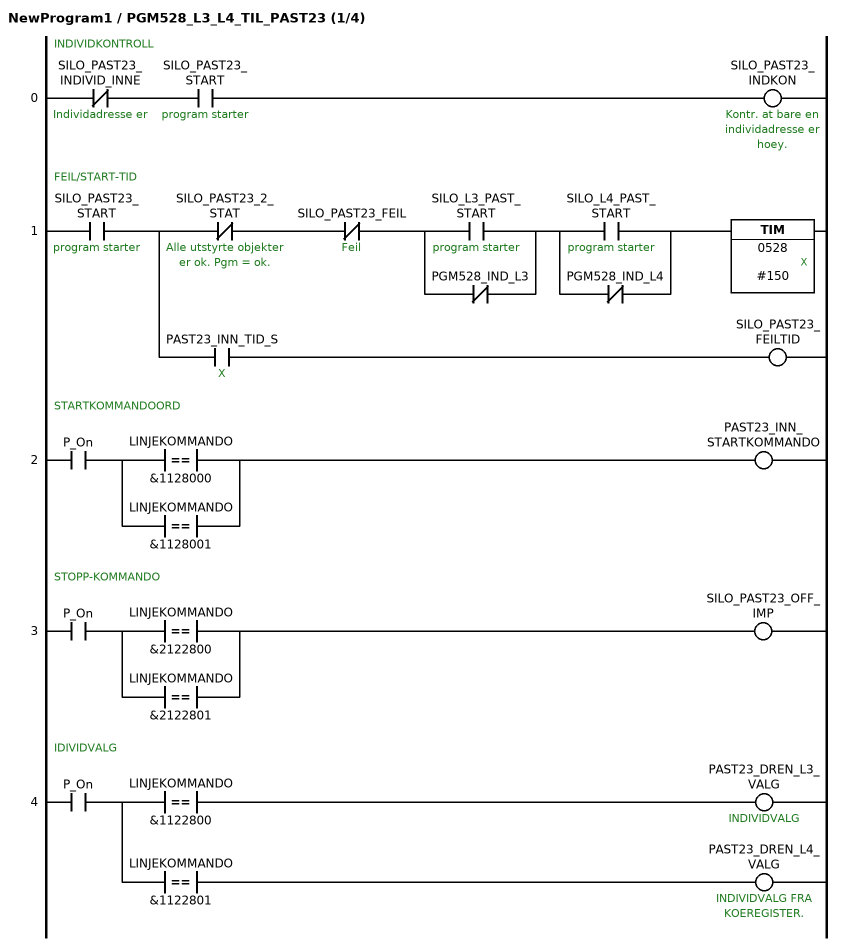
; [picture p696: NewProgram1 / PGM528_L3_L4_TIL_PAST23, rungs 0-4]
; rung 0: INDIVIDKONTROLL
LDNOT SILO_PAST23_INDIVID_INNE  ; Individadresse er
AND SILO_PAST23_START  ; program starter
OUT SILO_PAST23_INDKON  ; Kontr. at bare en individadresse er hoey.
; rung 1: FEIL/START-TID
LD SILO_PAST23_START  ; program starter
OUT TR0
ANDNOT SILO_PAST23_2_STAT  ; Alle utstyrte objekter er ok. Pgm = ok.
ANDNOT SILO_PAST23_FEIL  ; Feil
LD SILO_L3_PAST_START  ; program starter
ORNOT PGM528_IND_L3
ANDLD
LD SILO_L4_PAST_START  ; program starter
ORNOT PGM528_IND_L4
ANDLD
TIM 0528 #150  ; X
LD TR0
AND PAST23_INN_TID_S  ; X
OUT SILO_PAST23_FEILTID
; rung 2: STARTKOMMANDOORD
LD P_On
LD=L(301) LINJEKOMMANDO &1128000
OR=L(301) LINJEKOMMANDO &1128001
ANDLD
OUT PAST23_INN_STARTKOMMANDO
; rung 3: STOPP-KOMMANDO
LD P_On
LD=L(301) LINJEKOMMANDO &2122800
OR=L(301) LINJEKOMMANDO &2122801
ANDLD
OUT SILO_PAST23_OFF_IMP
; rung 4: IDIVIDVALG
LD P_On
OUT TR0
AND=L(301) LINJEKOMMANDO &1122800
OUT PAST23_DREN_L3_VALG  ; INDIVIDVALG
LD TR0
AND=L(301) LINJEKOMMANDO &1122801
OUT PAST23_DREN_L4_VALG  ; INDIVIDVALG FRA KOEREGISTER.

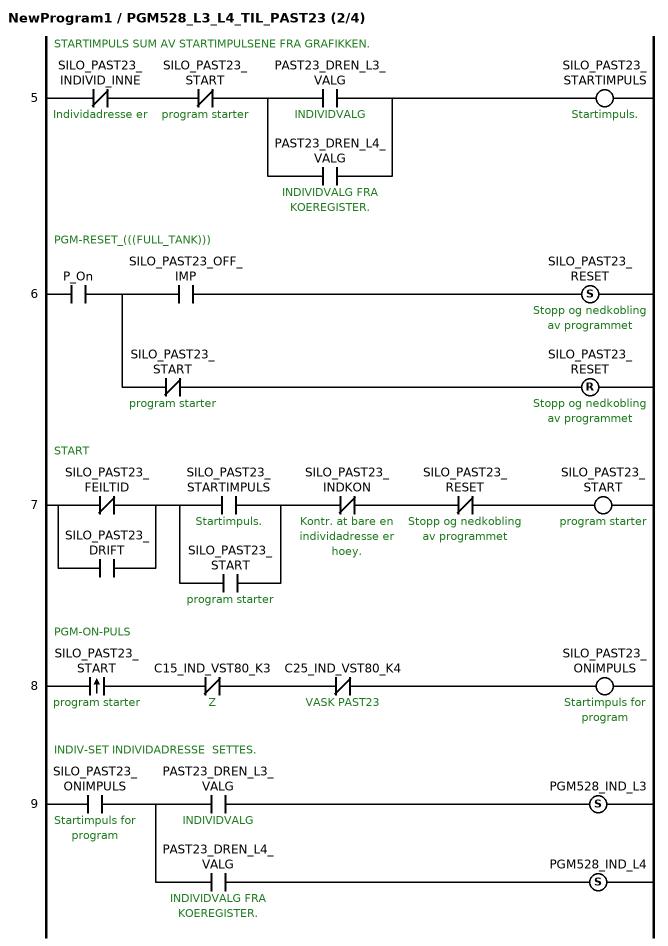
; rung 5: STARTIMPULS SUM AV STARTIMPULSENE FRA GRAFIKKEN.
LDNOT SILO_PAST23_INDIVID_INNE  ; Individadresse er
ANDNOT SILO_PAST23_START  ; program starter
LD PAST23_DREN_L3_VALG  ; INDIVIDVALG
OR PAST23_DREN_L4_VALG  ; INDIVIDVALG FRA KOEREGISTER.
ANDLD
OUT SILO_PAST23_STARTIMPULS  ; Startimpuls.
; rung 6: PGM-RESET_(((FULL_TANK)))
LD P_On
OUT TR0
AND SILO_PAST23_OFF_IMP
SET SILO_PAST23_RESET  ; Stopp og nedkobling av programmet
LD TR0
ANDNOT SILO_PAST23_START  ; program starter
RSET SILO_PAST23_RESET  ; Stopp og nedkobling av programmet
; rung 7: START
LDNOT SILO_PAST23_FEILTID
OR SILO_PAST23_DRIFT
LD SILO_PAST23_STARTIMPULS  ; Startimpuls.
OR SILO_PAST23_START  ; program starter
ANDLD
ANDNOT SILO_PAST23_INDKON  ; Kontr. at bare en individadresse er hoey.
ANDNOT SILO_PAST23_RESET  ; Stopp og nedkobling av programmet
OUT SILO_PAST23_START  ; program starter
; rung 8: PGM-ON-PULS
@LD SILO_PAST23_START  ; program starter
ANDNOT C15_IND_VST80_K3  ; Z
ANDNOT C25_IND_VST80_K4  ; VASK PAST23
OUT SILO_PAST23_ONIMPULS  ; Startimpuls for  program
; rung 9: INDIV-SET INDIVIDADRESSE  SETTES.
LD SILO_PAST23_ONIMPULS  ; Startimpuls for  program
OUT TR0
AND PAST23_DREN_L3_VALG  ; INDIVIDVALG
SET PGM528_IND_L3
LD TR0
AND PAST23_DREN_L4_VALG  ; INDIVIDVALG FRA KOEREGISTER.
SET PGM528_IND_L4

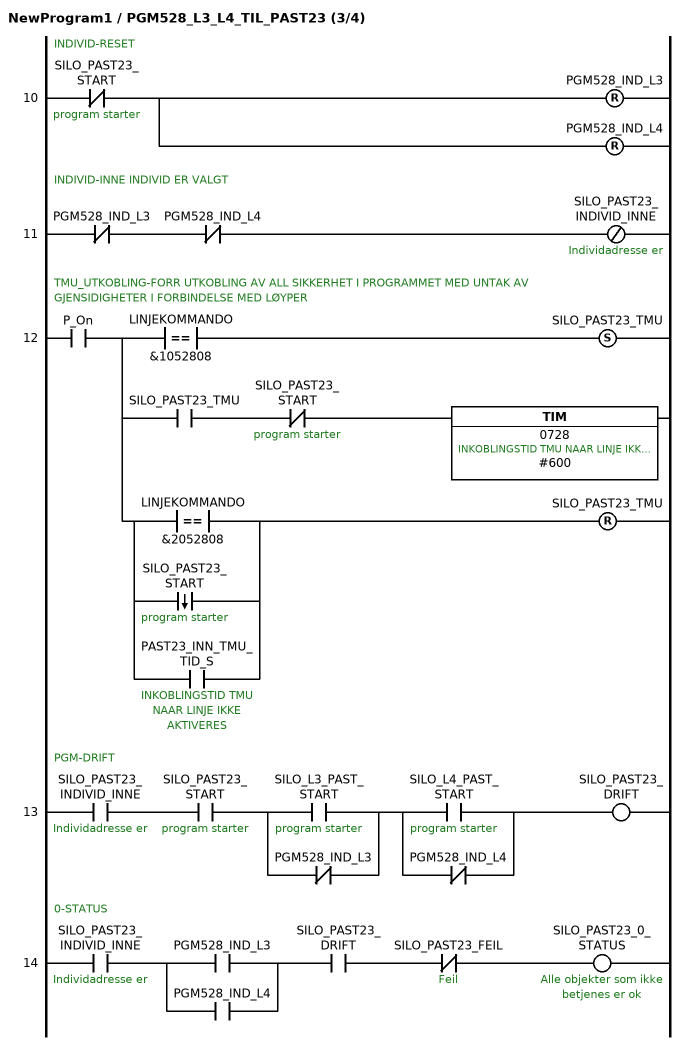
; rung 10: INDIVID-RESET
LDNOT SILO_PAST23_START  ; program starter
RSET PGM528_IND_L3
RSET PGM528_IND_L4
; rung 11: INDIVID-INNE INDIVID ER VALGT
LDNOT PGM528_IND_L3
ANDNOT PGM528_IND_L4
OUTNOT SILO_PAST23_INDIVID_INNE  ; Individadresse er
; rung 12: TMU_UTKOBLING-FORR UTKOBLING AV ALL SIKKERHET I PROGRAMMET MED UNTAK AV GJENSIDIGHETER I FORBINDELSE MED LØYPER
LD P_On
OUT TR0
AND=L(301) LINJEKOMMANDO &1052808
SET SILO_PAST23_TMU
LD TR0
AND SILO_PAST23_TMU
ANDNOT SILO_PAST23_START  ; program starter
TIM 0728 #600  ; INKOBLINGSTID TMU NAAR LINJE IKKE AKTIVERES
LD TR0
LD=L(301) LINJEKOMMANDO &2052808
%OR SILO_PAST23_START  ; program starter
OR PAST23_INN_TMU_TID_S  ; INKOBLINGSTID TMU NAAR LINJE IKKE AKTIVERES
ANDLD
RSET SILO_PAST23_TMU
; rung 13: PGM-DRIFT
LD SILO_PAST23_INDIVID_INNE  ; Individadresse er
AND SILO_PAST23_START  ; program starter
LD SILO_L3_PAST_START  ; program starter
ORNOT PGM528_IND_L3
ANDLD
LD SILO_L4_PAST_START  ; program starter
ORNOT PGM528_IND_L4
ANDLD
OUT SILO_PAST23_DRIFT
; rung 14: 0-STATUS
LD SILO_PAST23_INDIVID_INNE  ; Individadresse er
LD PGM528_IND_L3
OR PGM528_IND_L4
ANDLD
AND SILO_PAST23_DRIFT
ANDNOT SILO_PAST23_FEIL  ; Feil
OUT SILO_PAST23_0_STATUS  ; Alle objekter som ikke betjenes er ok

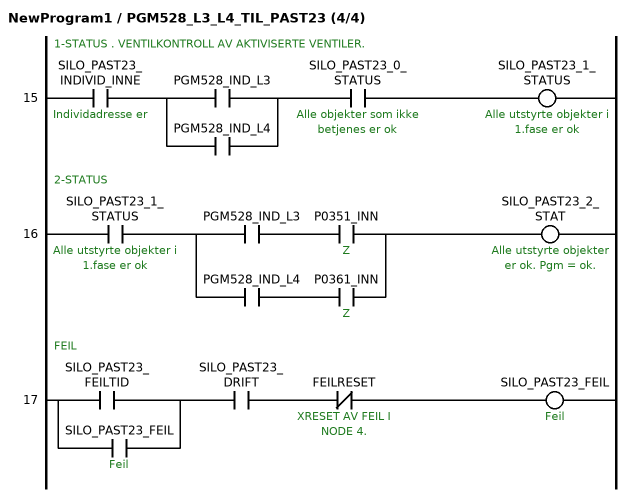
; rung 15: 1-STATUS . VENTILKONTROLL AV AKTIVISERTE VENTILER.
LD SILO_PAST23_INDIVID_INNE  ; Individadresse er
LD PGM528_IND_L3
OR PGM528_IND_L4
ANDLD
AND SILO_PAST23_0_STATUS  ; Alle objekter som ikke betjenes er ok
OUT SILO_PAST23_1_STATUS  ; Alle utstyrte objekter i 1.fase er ok
; rung 16: 2-STATUS
LD SILO_PAST23_1_STATUS  ; Alle utstyrte objekter i 1.fase er ok
LD PGM528_IND_L3
AND P0351_INN  ; Z
LD PGM528_IND_L4
AND P0361_INN  ; Z
ORLD
ANDLD
OUT SILO_PAST23_2_STAT  ; Alle utstyrte objekter er ok. Pgm = ok.
; rung 17: FEIL
LD SILO_PAST23_FEILTID
OR SILO_PAST23_FEIL  ; Feil
AND SILO_PAST23_DRIFT
ANDNOT FEILRESET  ; XRESET AV FEIL I NODE 4.
OUT SILO_PAST23_FEIL  ; Feil

### Section PGM529_T24_CONTAINER_TIL_PAST23

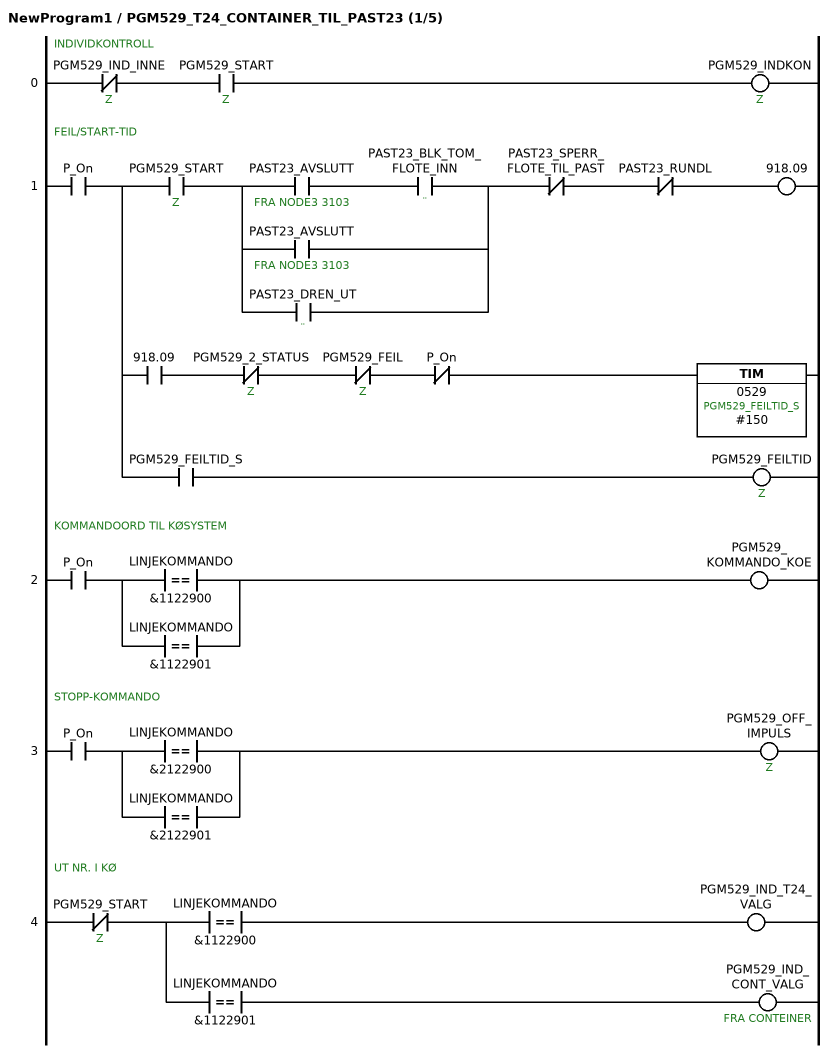
; rung 0: INDIVIDKONTROLL
LDNOT PGM529_IND_INNE  ; Z
AND PGM529_START  ; Z
OUT PGM529_INDKON  ; Z
; rung 1: FEIL/START-TID
LD P_On
OUT TR0
AND PGM529_START  ; Z
LD PAST23_AVSLUTT  ; FRA NODE3 3103
AND PAST23_BLK_TOM_FLOTE_INN  ; ¨
OR PAST23_AVSLUTT  ; FRA NODE3 3103
OR PAST23_DREN_UT  ; ¨
ANDLD
ANDNOT PAST23_SPERR_FLOTE_TIL_PAST
ANDNOT PAST23_RUNDL
OUT 918.09
LD TR0
AND 918.09
ANDNOT PGM529_2_STATUS  ; Z
ANDNOT PGM529_FEIL  ; Z
ANDNOT P_On
TIM 0529 #150  ; PGM529_FEILTID_S
LD TR0
AND PGM529_FEILTID_S
OUT PGM529_FEILTID  ; Z
; rung 2: KOMMANDOORD TIL KØSYSTEM
LD P_On
LD=L(301) LINJEKOMMANDO &1122900
OR=L(301) LINJEKOMMANDO &1122901
ANDLD
OUT PGM529_KOMMANDO_KOE
; rung 3: STOPP-KOMMANDO
LD P_On
LD=L(301) LINJEKOMMANDO &2122900
OR=L(301) LINJEKOMMANDO &2122901
ANDLD
OUT PGM529_OFF_IMPULS  ; Z
; rung 4: UT NR. I KØ
LDNOT PGM529_START  ; Z
OUT TR0
AND=L(301) LINJEKOMMANDO &1122900
OUT PGM529_IND_T24_VALG
LD TR0
AND=L(301) LINJEKOMMANDO &1122901
OUT PGM529_IND_CONT_VALG  ; FRA CONTEINER

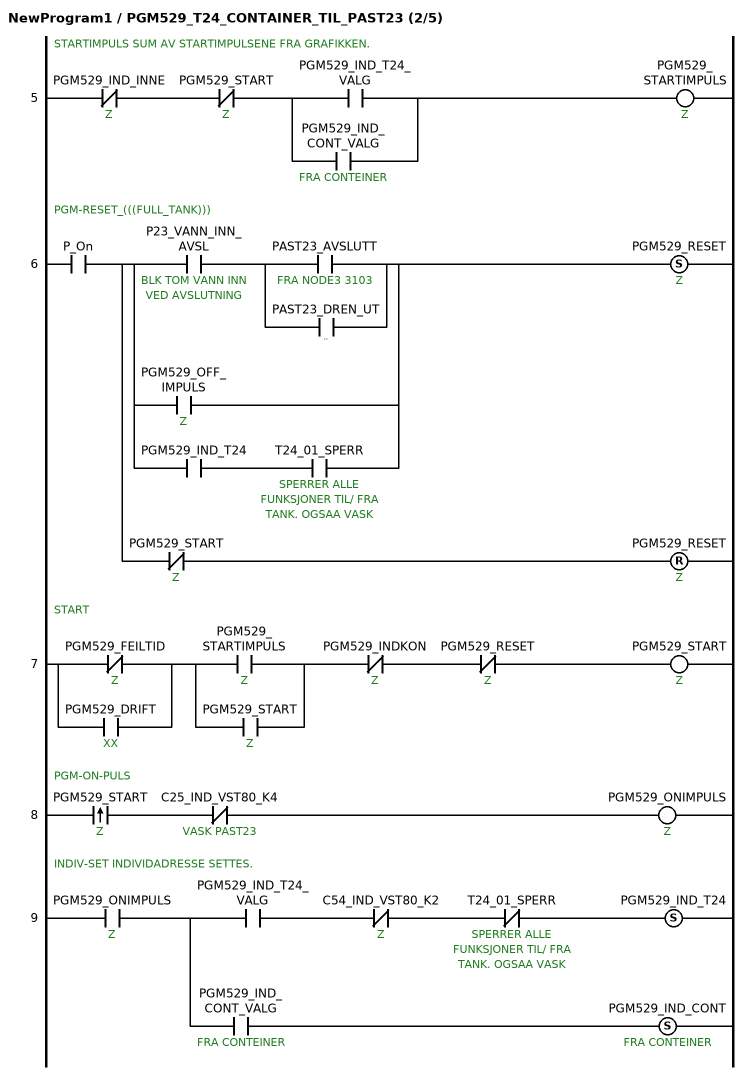
; rung 5: STARTIMPULS SUM AV STARTIMPULSENE FRA GRAFIKKEN.
LDNOT PGM529_IND_INNE  ; Z
ANDNOT PGM529_START  ; Z
LD PGM529_IND_T24_VALG
OR PGM529_IND_CONT_VALG  ; FRA CONTEINER
ANDLD
OUT PGM529_STARTIMPULS  ; Z
; rung 6: PGM-RESET_(((FULL_TANK)))
LD P_On
OUT TR0
LD P23_VANN_INN_AVSL  ; BLK TOM VANN INN VED AVSLUTNING
LD PAST23_AVSLUTT  ; FRA NODE3 3103
OR PAST23_DREN_UT  ; ¨
ANDLD
OR PGM529_OFF_IMPULS  ; Z
LD PGM529_IND_T24
AND T24_01_SPERR  ; SPERRER ALLE FUNKSJONER TIL/ FRA TANK. OGSAA VASK
ORLD
ANDLD
SET PGM529_RESET  ; Z
LD TR0
ANDNOT PGM529_START  ; Z
RSET PGM529_RESET  ; Z
; rung 7: START
LDNOT PGM529_FEILTID  ; Z
OR PGM529_DRIFT  ; XX
LD PGM529_STARTIMPULS  ; Z
OR PGM529_START  ; Z
ANDLD
ANDNOT PGM529_INDKON  ; Z
ANDNOT PGM529_RESET  ; Z
OUT PGM529_START  ; Z
; rung 8: PGM-ON-PULS
@LD PGM529_START  ; Z
ANDNOT C25_IND_VST80_K4  ; VASK PAST23
OUT PGM529_ONIMPULS  ; Z
; rung 9: INDIV-SET INDIVIDADRESSE SETTES.
LD PGM529_ONIMPULS  ; Z
OUT TR0
AND PGM529_IND_T24_VALG
ANDNOT C54_IND_VST80_K2  ; Z
ANDNOT T24_01_SPERR  ; SPERRER ALLE FUNKSJONER TIL/ FRA TANK. OGSAA VASK
SET PGM529_IND_T24
LD TR0
AND PGM529_IND_CONT_VALG  ; FRA CONTEINER
SET PGM529_IND_CONT  ; FRA CONTEINER

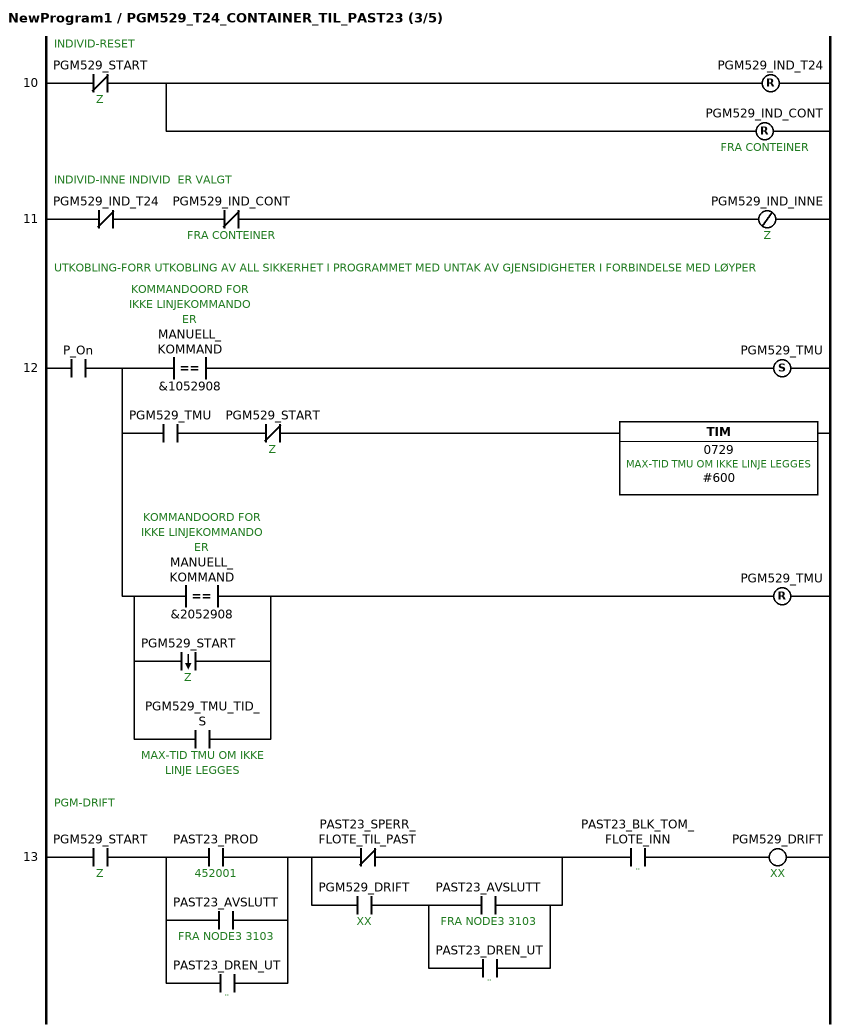
; rung 10: INDIVID-RESET
LDNOT PGM529_START  ; Z
RSET PGM529_IND_T24
RSET PGM529_IND_CONT  ; FRA CONTEINER
; rung 11: INDIVID-INNE INDIVID  ER VALGT
LDNOT PGM529_IND_T24
ANDNOT PGM529_IND_CONT  ; FRA CONTEINER
OUTNOT PGM529_IND_INNE  ; Z
; rung 12: UTKOBLING-FORR UTKOBLING AV ALL SIKKERHET I PROGRAMMET MED UNTAK AV GJENSIDIGHETER I FORBINDELSE MED LØYPER
LD P_On
OUT TR0
AND=L(301) MANUELL_KOMMAND &1052908  ; KOMMANDOORD FOR IKKE LINJEKOMMANDOER
SET PGM529_TMU
LD TR0
AND PGM529_TMU
ANDNOT PGM529_START  ; Z
TIM 0729 #600  ; MAX-TID TMU OM IKKE LINJE LEGGES
LD TR0
LD=L(301) MANUELL_KOMMAND &2052908  ; KOMMANDOORD FOR IKKE LINJEKOMMANDOER
%OR PGM529_START  ; Z
OR PGM529_TMU_TID_S  ; MAX-TID TMU OM IKKE LINJE LEGGES
ANDLD
RSET PGM529_TMU
; rung 13: PGM-DRIFT
LD PGM529_START  ; Z
LD PAST23_PROD  ; 452001
OR PAST23_AVSLUTT  ; FRA NODE3 3103
OR PAST23_DREN_UT  ; ¨
ANDLD
LDNOT PAST23_SPERR_FLOTE_TIL_PAST
LD PGM529_DRIFT  ; XX
LD PAST23_AVSLUTT  ; FRA NODE3 3103
OR PAST23_DREN_UT  ; ¨
ANDLD
ORLD
ANDLD
AND PAST23_BLK_TOM_FLOTE_INN  ; ¨
OUT PGM529_DRIFT  ; XX

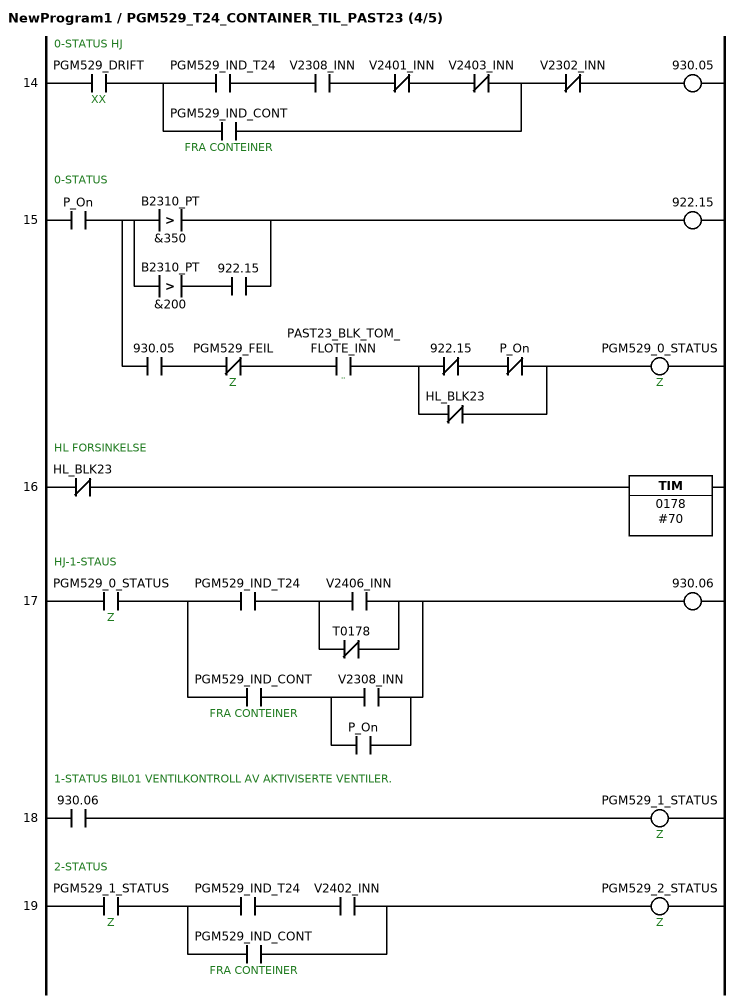
; rung 14: 0-STATUS HJ
LD PGM529_DRIFT  ; XX
LD PGM529_IND_T24
AND V2308_INN
ANDNOT V2401_INN
ANDNOT V2403_INN
OR PGM529_IND_CONT  ; FRA CONTEINER
ANDLD
ANDNOT V2302_INN
OUT 930.05
; rung 15: 0-STATUS
LD P_On
OUT TR0
LD>(320) B2310_PT &350
LD>(320) B2310_PT &200
AND 922.15
ORLD
ANDLD
OUT 922.15
LD TR0
AND 930.05
ANDNOT PGM529_FEIL  ; Z
AND PAST23_BLK_TOM_FLOTE_INN  ; ¨
LDNOT 922.15
ANDNOT P_On
ORNOT HL_BLK23
ANDLD
OUT PGM529_0_STATUS  ; Z
; rung 16: HL FORSINKELSE
LDNOT HL_BLK23
TIM 0178 #70
; rung 17: HJ-1-STAUS
LD PGM529_0_STATUS  ; Z
LD PGM529_IND_T24
LD V2406_INN
ORNOT T0178
ANDLD
LD PGM529_IND_CONT  ; FRA CONTEINER
LD V2308_INN
OR P_On
ANDLD
ORLD
ANDLD
OUT 930.06
; rung 18: 1-STATUS BIL01 VENTILKONTROLL AV AKTIVISERTE VENTILER.
LD 930.06
OUT PGM529_1_STATUS  ; Z
; rung 19: 2-STATUS
LD PGM529_1_STATUS  ; Z
LD PGM529_IND_T24
AND V2402_INN
OR PGM529_IND_CONT  ; FRA CONTEINER
ANDLD
OUT PGM529_2_STATUS  ; Z

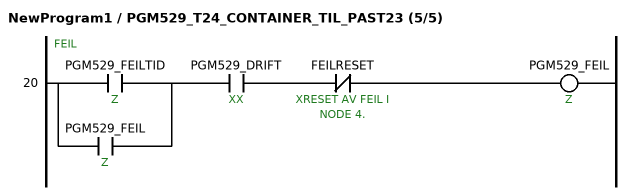
; rung 20: FEIL
LD PGM529_FEILTID  ; Z
OR PGM529_FEIL  ; Z
AND PGM529_DRIFT  ; XX
ANDNOT FEILRESET  ; XRESET AV FEIL I NODE 4.
OUT PGM529_FEIL  ; Z

### Section PGM584_TIL_T2740_2741

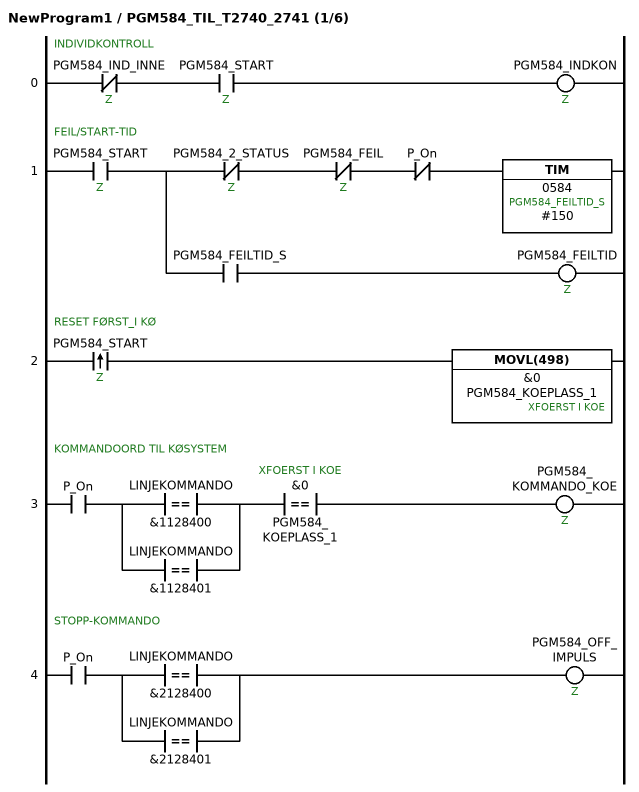
; rung 0: INDIVIDKONTROLL
LDNOT PGM584_IND_INNE  ; Z
AND PGM584_START  ; Z
OUT PGM584_INDKON  ; Z
; rung 1: FEIL/START-TID
LD PGM584_START  ; Z
OUT TR0
ANDNOT PGM584_2_STATUS  ; Z
ANDNOT PGM584_FEIL  ; Z
ANDNOT P_On
TIM 0584 #150  ; PGM584_FEILTID_S
LD TR0
AND PGM584_FEILTID_S
OUT PGM584_FEILTID  ; Z
; rung 2: RESET FØRST_I KØ
@LD PGM584_START  ; Z
MOVL(498) &0 PGM584_KOEPLASS_1  ; XFOERST I KOE
; rung 3: KOMMANDOORD TIL KØSYSTEM
LD P_On
LD=L(301) LINJEKOMMANDO &1128400
OR=L(301) LINJEKOMMANDO &1128401
ANDLD
AND=L(301) &0 PGM584_KOEPLASS_1  ; XFOERST I KOE
OUT PGM584_KOMMANDO_KOE  ; Z
; rung 4: STOPP-KOMMANDO
LD P_On
LD=L(301) LINJEKOMMANDO &2128400
OR=L(301) LINJEKOMMANDO &2128401
ANDLD
OUT PGM584_OFF_IMPULS  ; Z

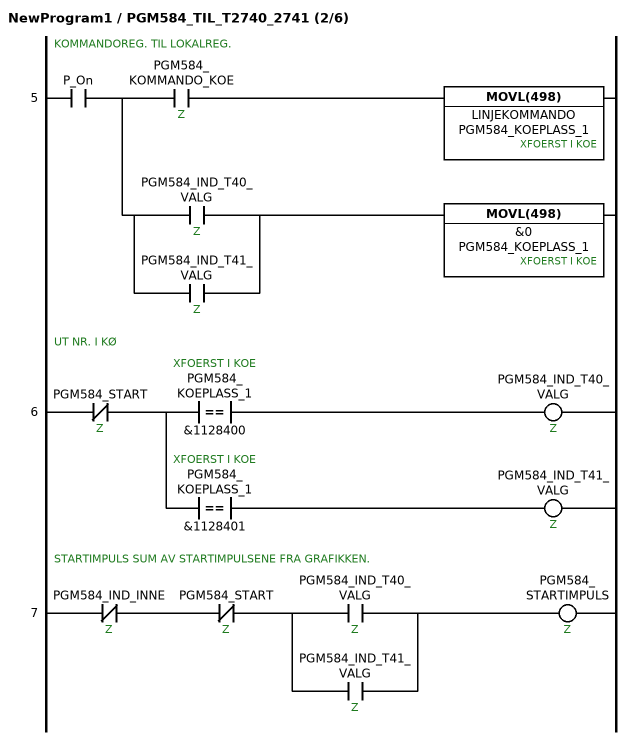
; rung 5: KOMMANDOREG. TIL LOKALREG.
LD P_On
OUT TR0
AND PGM584_KOMMANDO_KOE  ; Z
MOVL(498) LINJEKOMMANDO PGM584_KOEPLASS_1  ; XFOERST I KOE
LD TR0
LD PGM584_IND_T40_VALG  ; Z
OR PGM584_IND_T41_VALG  ; Z
ANDLD
MOVL(498) &0 PGM584_KOEPLASS_1  ; XFOERST I KOE
; rung 6: UT NR. I KØ
LDNOT PGM584_START  ; Z
OUT TR0
AND=L(301) PGM584_KOEPLASS_1 &1128400  ; XFOERST I KOE
OUT PGM584_IND_T40_VALG  ; Z
LD TR0
AND=L(301) PGM584_KOEPLASS_1 &1128401  ; XFOERST I KOE
OUT PGM584_IND_T41_VALG  ; Z
; rung 7: STARTIMPULS SUM AV STARTIMPULSENE FRA GRAFIKKEN.
LDNOT PGM584_IND_INNE  ; Z
ANDNOT PGM584_START  ; Z
LD PGM584_IND_T40_VALG  ; Z
OR PGM584_IND_T41_VALG  ; Z
ANDLD
OUT PGM584_STARTIMPULS  ; Z

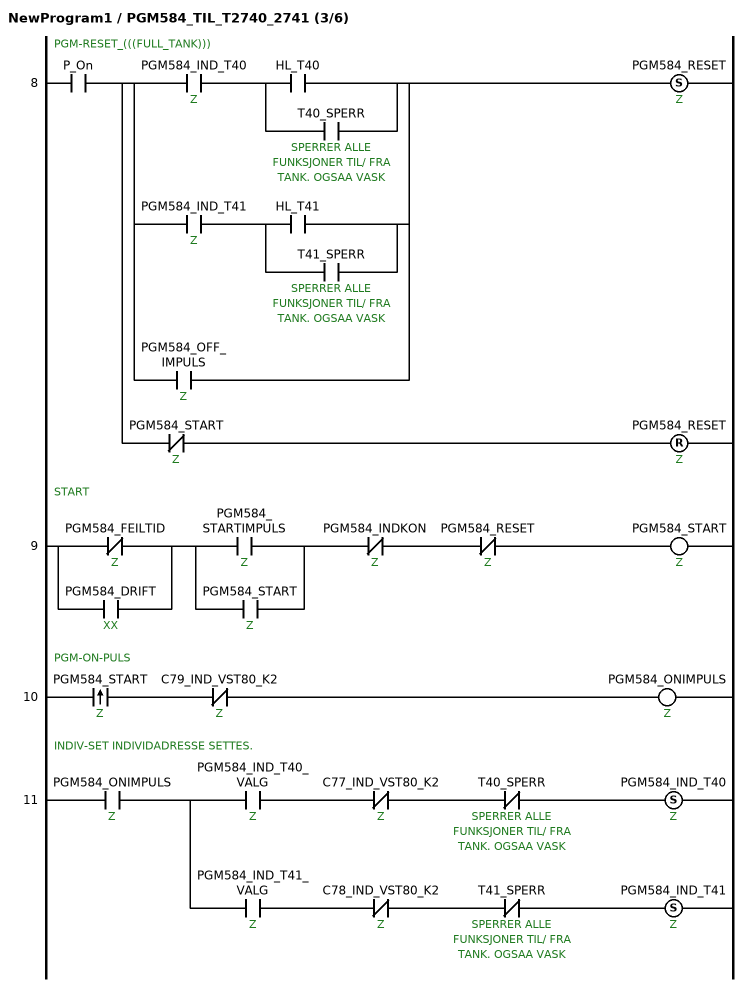
; rung 8: PGM-RESET_(((FULL_TANK)))
LD P_On
OUT TR0
LD PGM584_IND_T40  ; Z
LD HL_T40
OR T40_SPERR  ; SPERRER ALLE FUNKSJONER TIL/ FRA TANK. OGSAA VASK
ANDLD
LD PGM584_IND_T41  ; Z
LD HL_T41
OR T41_SPERR  ; SPERRER ALLE FUNKSJONER TIL/ FRA TANK. OGSAA VASK
ANDLD
ORLD
OR PGM584_OFF_IMPULS  ; Z
ANDLD
SET PGM584_RESET  ; Z
LD TR0
ANDNOT PGM584_START  ; Z
RSET PGM584_RESET  ; Z
; rung 9: START
LDNOT PGM584_FEILTID  ; Z
OR PGM584_DRIFT  ; XX
LD PGM584_STARTIMPULS  ; Z
OR PGM584_START  ; Z
ANDLD
ANDNOT PGM584_INDKON  ; Z
ANDNOT PGM584_RESET  ; Z
OUT PGM584_START  ; Z
; rung 10: PGM-ON-PULS
@LD PGM584_START  ; Z
ANDNOT C79_IND_VST80_K2  ; Z
OUT PGM584_ONIMPULS  ; Z
; rung 11: INDIV-SET INDIVIDADRESSE SETTES.
LD PGM584_ONIMPULS  ; Z
OUT TR0
AND PGM584_IND_T40_VALG  ; Z
ANDNOT C77_IND_VST80_K2  ; Z
ANDNOT T40_SPERR  ; SPERRER ALLE FUNKSJONER TIL/ FRA TANK. OGSAA VASK
SET PGM584_IND_T40  ; Z
LD TR0
AND PGM584_IND_T41_VALG  ; Z
ANDNOT C78_IND_VST80_K2  ; Z
ANDNOT T41_SPERR  ; SPERRER ALLE FUNKSJONER TIL/ FRA TANK. OGSAA VASK
SET PGM584_IND_T41  ; Z

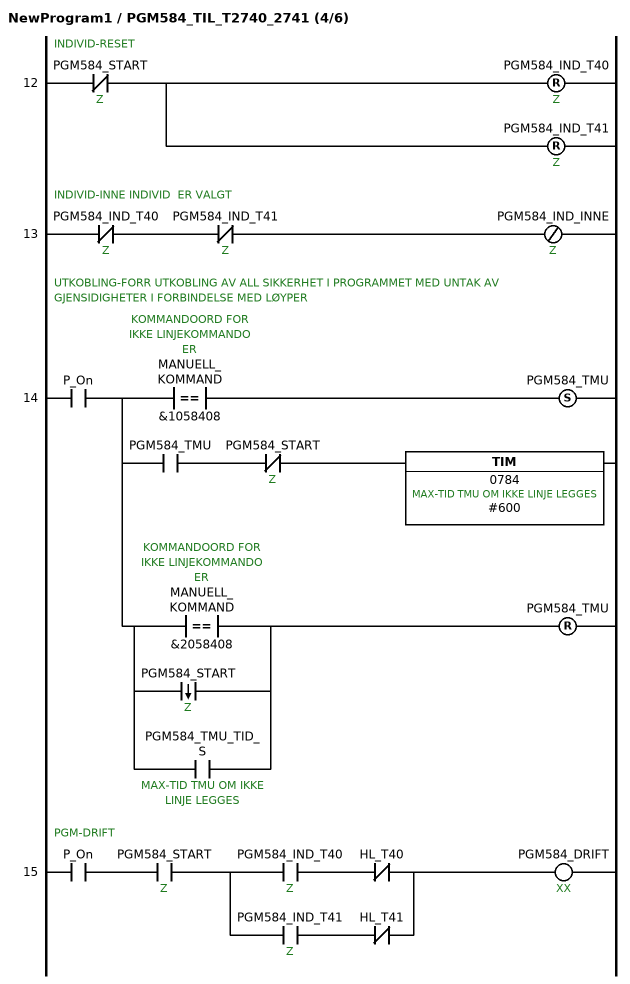
; rung 12: INDIVID-RESET
LDNOT PGM584_START  ; Z
RSET PGM584_IND_T40  ; Z
RSET PGM584_IND_T41  ; Z
; rung 13: INDIVID-INNE INDIVID  ER VALGT
LDNOT PGM584_IND_T40  ; Z
ANDNOT PGM584_IND_T41  ; Z
OUTNOT PGM584_IND_INNE  ; Z
; rung 14: UTKOBLING-FORR UTKOBLING AV ALL SIKKERHET I PROGRAMMET MED UNTAK AV GJENSIDIGHETER I FORBINDELSE MED LØYPER
LD P_On
OUT TR0
AND=L(301) MANUELL_KOMMAND &1058408  ; KOMMANDOORD FOR IKKE LINJEKOMMANDOER
SET PGM584_TMU
LD TR0
AND PGM584_TMU
ANDNOT PGM584_START  ; Z
TIM 0784 #600  ; MAX-TID TMU OM IKKE LINJE LEGGES
LD TR0
LD=L(301) MANUELL_KOMMAND &2058408  ; KOMMANDOORD FOR IKKE LINJEKOMMANDOER
%OR PGM584_START  ; Z
OR PGM584_TMU_TID_S  ; MAX-TID TMU OM IKKE LINJE LEGGES
ANDLD
RSET PGM584_TMU
; rung 15: PGM-DRIFT
LD P_On
AND PGM584_START  ; Z
LD PGM584_IND_T40  ; Z
ANDNOT HL_T40
LD PGM584_IND_T41  ; Z
ANDNOT HL_T41
ORLD
ANDLD
OUT PGM584_DRIFT  ; XX

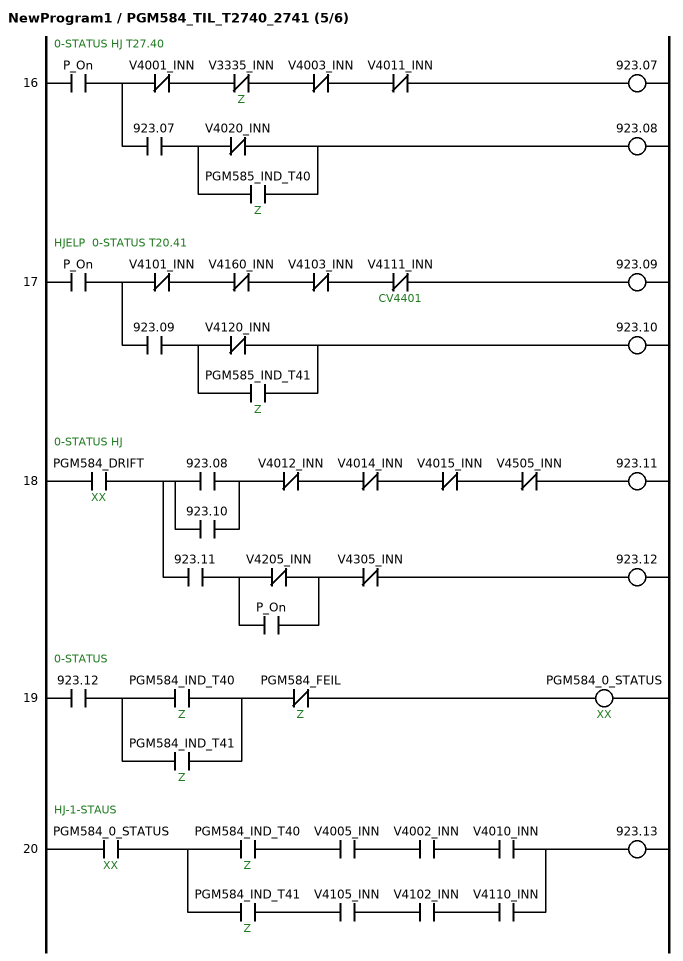
; rung 16: 0-STATUS HJ T27.40
LD P_On
OUT TR0
ANDNOT V4001_INN
ANDNOT V3335_INN  ; Z
ANDNOT V4003_INN
ANDNOT V4011_INN
OUT 923.07
LD TR0
AND 923.07
LDNOT V4020_INN
OR PGM585_IND_T40  ; Z
ANDLD
OUT 923.08
; rung 17: HJELP  0-STATUS T20.41
LD P_On
OUT TR0
ANDNOT V4101_INN
ANDNOT V4160_INN
ANDNOT V4103_INN
ANDNOT V4111_INN  ; CV4401
OUT 923.09
LD TR0
AND 923.09
LDNOT V4120_INN
OR PGM585_IND_T41  ; Z
ANDLD
OUT 923.10
; rung 18: 0-STATUS HJ
LD PGM584_DRIFT  ; XX
OUT TR0
LD 923.08
OR 923.10
ANDLD
ANDNOT V4012_INN
ANDNOT V4014_INN
ANDNOT V4015_INN
ANDNOT V4505_INN
OUT 923.11
LD TR0
AND 923.11
LDNOT V4205_INN
OR P_On
ANDLD
ANDNOT V4305_INN
OUT 923.12
; rung 19: 0-STATUS
LD 923.12
LD PGM584_IND_T40  ; Z
OR PGM584_IND_T41  ; Z
ANDLD
ANDNOT PGM584_FEIL  ; Z
OUT PGM584_0_STATUS  ; XX
; rung 20: HJ-1-STAUS
LD PGM584_0_STATUS  ; XX
LD PGM584_IND_T40  ; Z
AND V4005_INN
AND V4002_INN
AND V4010_INN
LD PGM584_IND_T41  ; Z
AND V4105_INN
AND V4102_INN
AND V4110_INN
ORLD
ANDLD
OUT 923.13

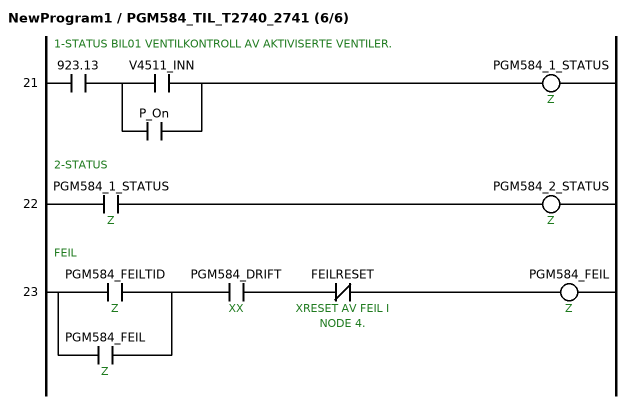
; rung 21: 1-STATUS BIL01 VENTILKONTROLL AV AKTIVISERTE VENTILER.
LD 923.13
LD V4511_INN
OR P_On
ANDLD
OUT PGM584_1_STATUS  ; Z
; rung 22: 2-STATUS
LD PGM584_1_STATUS  ; Z
OUT PGM584_2_STATUS  ; Z
; rung 23: FEIL
LD PGM584_FEILTID  ; Z
OR PGM584_FEIL  ; Z
AND PGM584_DRIFT  ; XX
ANDNOT FEILRESET  ; XRESET AV FEIL I NODE 4.
OUT PGM584_FEIL  ; Z

### Section PGM585_FRA_T2740_2741

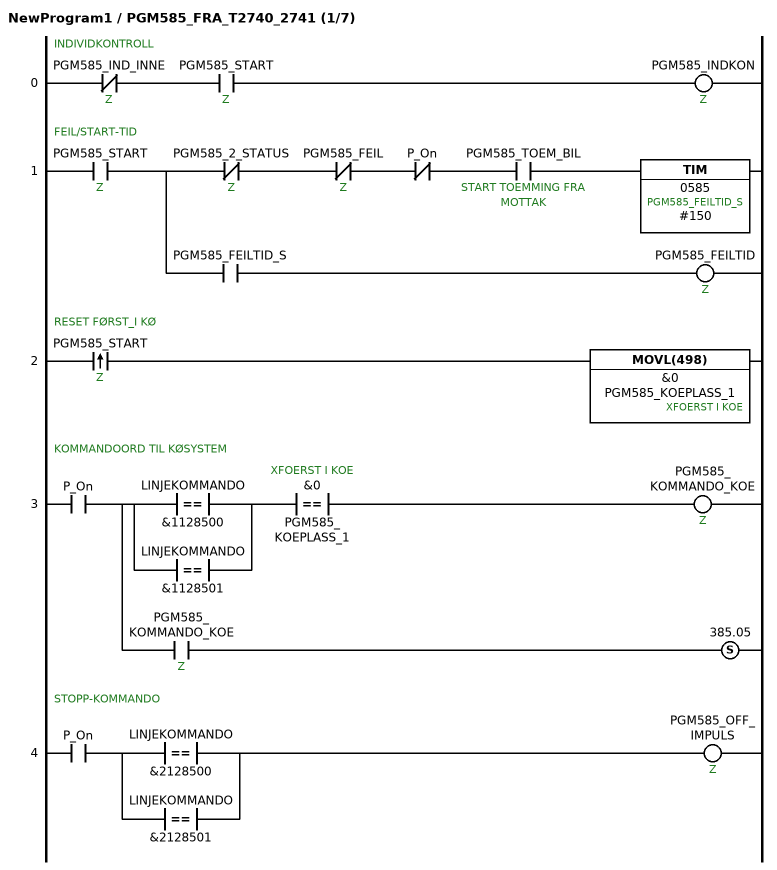
; rung 0: INDIVIDKONTROLL
LDNOT PGM585_IND_INNE  ; Z
AND PGM585_START  ; Z
OUT PGM585_INDKON  ; Z
; rung 1: FEIL/START-TID
LD PGM585_START  ; Z
OUT TR0
ANDNOT PGM585_2_STATUS  ; Z
ANDNOT PGM585_FEIL  ; Z
ANDNOT P_On
AND PGM585_TOEM_BIL  ; START TOEMMING FRA MOTTAK
TIM 0585 #150  ; PGM585_FEILTID_S
LD TR0
AND PGM585_FEILTID_S
OUT PGM585_FEILTID  ; Z
; rung 2: RESET FØRST_I KØ
@LD PGM585_START  ; Z
MOVL(498) &0 PGM585_KOEPLASS_1  ; XFOERST I KOE
; rung 3: KOMMANDOORD TIL KØSYSTEM
LD P_On
OUT TR0
LD=L(301) LINJEKOMMANDO &1128500
OR=L(301) LINJEKOMMANDO &1128501
ANDLD
AND=L(301) &0 PGM585_KOEPLASS_1  ; XFOERST I KOE
OUT PGM585_KOMMANDO_KOE  ; Z
LD TR0
AND PGM585_KOMMANDO_KOE  ; Z
SET 385.05
; rung 4: STOPP-KOMMANDO
LD P_On
LD=L(301) LINJEKOMMANDO &2128500
OR=L(301) LINJEKOMMANDO &2128501
ANDLD
OUT PGM585_OFF_IMPULS  ; Z

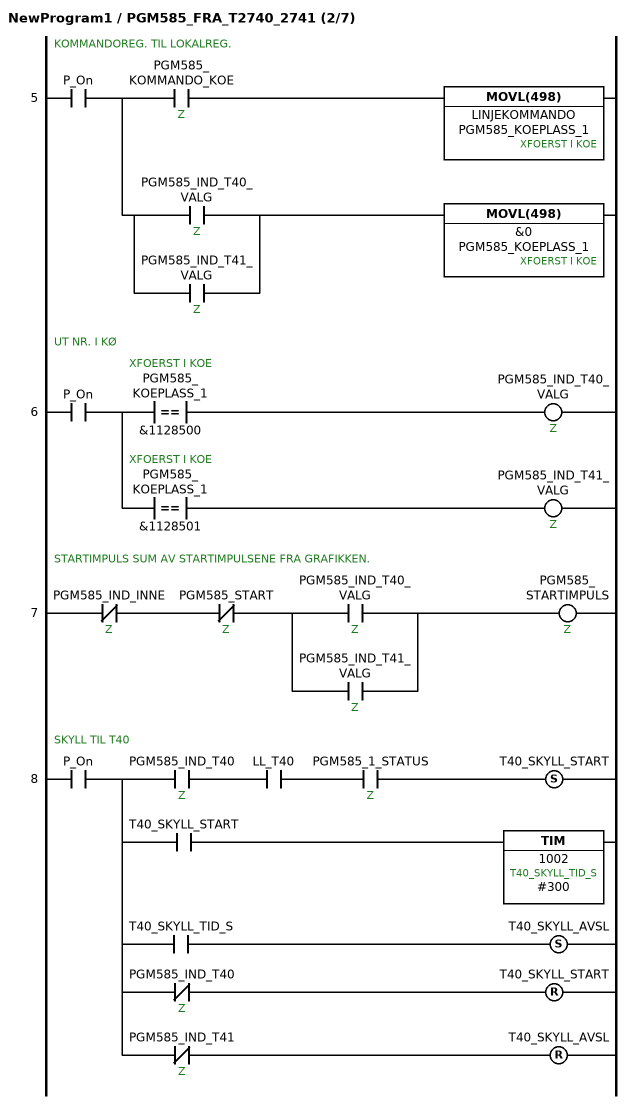
; rung 5: KOMMANDOREG. TIL LOKALREG.
LD P_On
OUT TR0
AND PGM585_KOMMANDO_KOE  ; Z
MOVL(498) LINJEKOMMANDO PGM585_KOEPLASS_1  ; XFOERST I KOE
LD TR0
LD PGM585_IND_T40_VALG  ; Z
OR PGM585_IND_T41_VALG  ; Z
ANDLD
MOVL(498) &0 PGM585_KOEPLASS_1  ; XFOERST I KOE
; rung 6: UT NR. I KØ
LD P_On
OUT TR0
AND=L(301) PGM585_KOEPLASS_1 &1128500  ; XFOERST I KOE
OUT PGM585_IND_T40_VALG  ; Z
LD TR0
AND=L(301) PGM585_KOEPLASS_1 &1128501  ; XFOERST I KOE
OUT PGM585_IND_T41_VALG  ; Z
; rung 7: STARTIMPULS SUM AV STARTIMPULSENE FRA GRAFIKKEN.
LDNOT PGM585_IND_INNE  ; Z
ANDNOT PGM585_START  ; Z
LD PGM585_IND_T40_VALG  ; Z
OR PGM585_IND_T41_VALG  ; Z
ANDLD
OUT PGM585_STARTIMPULS  ; Z
; rung 8: SKYLL TIL T40
LD P_On
OUT TR0
AND PGM585_IND_T40  ; Z
AND LL_T40
AND PGM585_1_STATUS  ; Z
SET T40_SKYLL_START
LD TR0
AND T40_SKYLL_START
TIM 1002 #300  ; T40_SKYLL_TID_S
LD TR0
AND T40_SKYLL_TID_S
SET T40_SKYLL_AVSL
LD TR0
ANDNOT PGM585_IND_T40  ; Z
RSET T40_SKYLL_START
LD TR0
ANDNOT PGM585_IND_T41  ; Z
RSET T40_SKYLL_AVSL

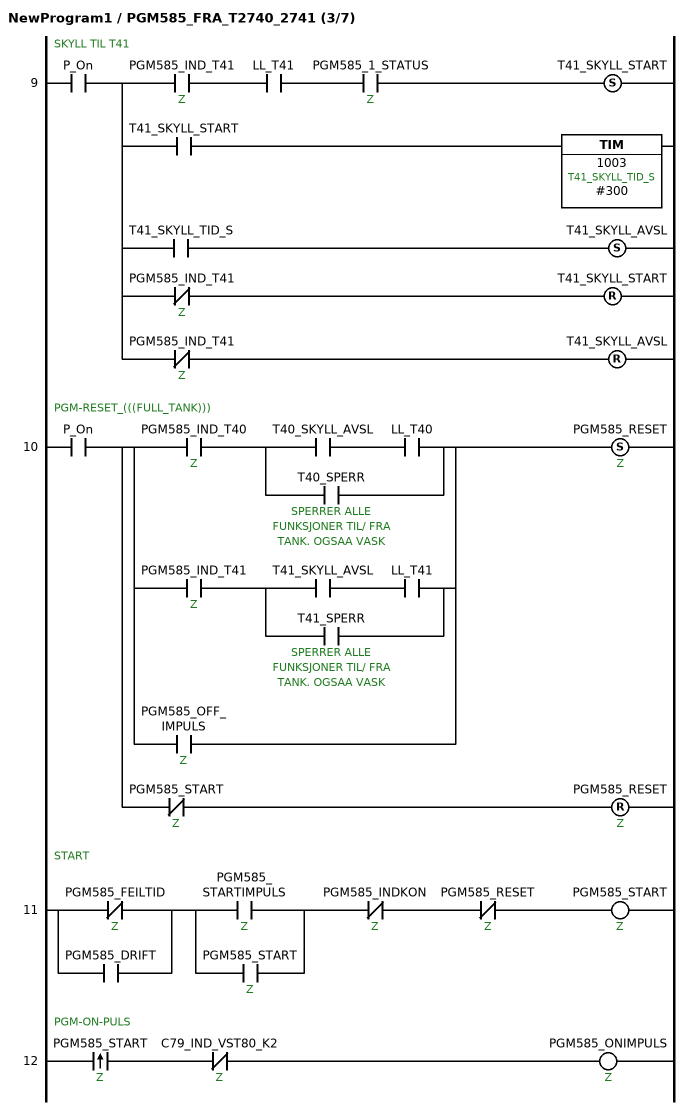
; rung 9: SKYLL TIL T41
LD P_On
OUT TR0
AND PGM585_IND_T41  ; Z
AND LL_T41
AND PGM585_1_STATUS  ; Z
SET T41_SKYLL_START
LD TR0
AND T41_SKYLL_START
TIM 1003 #300  ; T41_SKYLL_TID_S
LD TR0
AND T41_SKYLL_TID_S
SET T41_SKYLL_AVSL
LD TR0
ANDNOT PGM585_IND_T41  ; Z
RSET T41_SKYLL_START
LD TR0
ANDNOT PGM585_IND_T41  ; Z
RSET T41_SKYLL_AVSL
; rung 10: PGM-RESET_(((FULL_TANK)))
LD P_On
OUT TR0
LD PGM585_IND_T40  ; Z
LD T40_SKYLL_AVSL
AND LL_T40
OR T40_SPERR  ; SPERRER ALLE FUNKSJONER TIL/ FRA TANK. OGSAA VASK
ANDLD
LD PGM585_IND_T41  ; Z
LD T41_SKYLL_AVSL
AND LL_T41
OR T41_SPERR  ; SPERRER ALLE FUNKSJONER TIL/ FRA TANK. OGSAA VASK
ANDLD
ORLD
OR PGM585_OFF_IMPULS  ; Z
ANDLD
SET PGM585_RESET  ; Z
LD TR0
ANDNOT PGM585_START  ; Z
RSET PGM585_RESET  ; Z
; rung 11: START
LDNOT PGM585_FEILTID  ; Z
OR PGM585_DRIFT
LD PGM585_STARTIMPULS  ; Z
OR PGM585_START  ; Z
ANDLD
ANDNOT PGM585_INDKON  ; Z
ANDNOT PGM585_RESET  ; Z
OUT PGM585_START  ; Z
; rung 12: PGM-ON-PULS
@LD PGM585_START  ; Z
ANDNOT C79_IND_VST80_K2  ; Z
OUT PGM585_ONIMPULS  ; Z

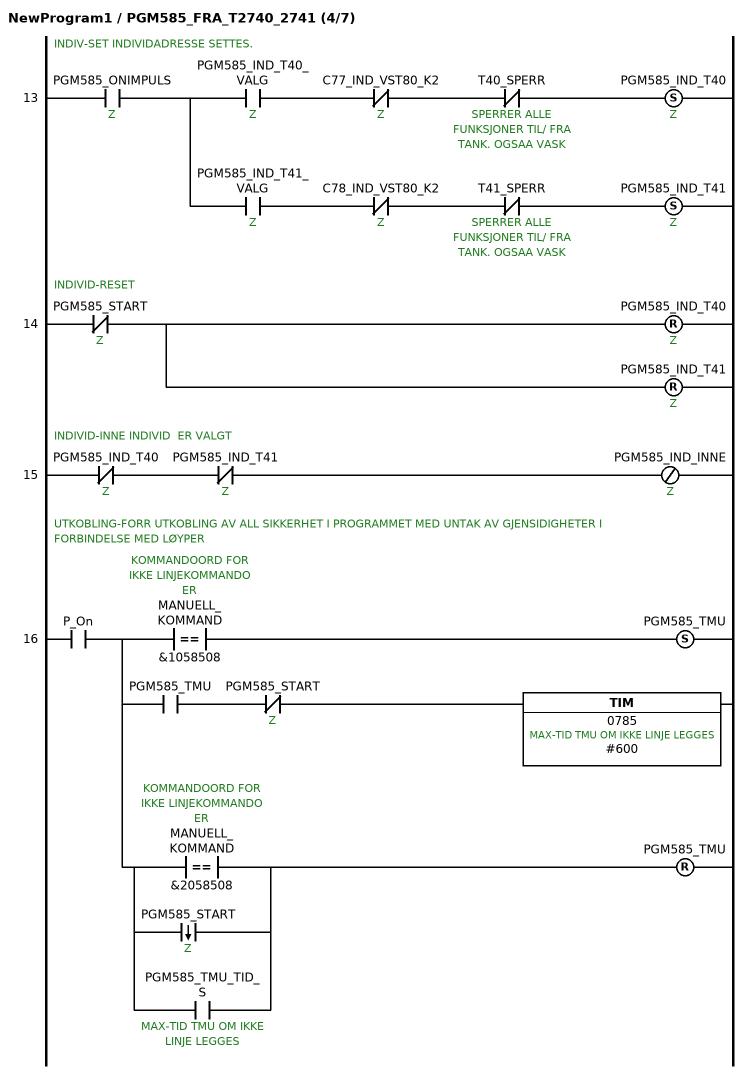
; rung 13: INDIV-SET INDIVIDADRESSE SETTES.
LD PGM585_ONIMPULS  ; Z
OUT TR0
AND PGM585_IND_T40_VALG  ; Z
ANDNOT C77_IND_VST80_K2  ; Z
ANDNOT T40_SPERR  ; SPERRER ALLE FUNKSJONER TIL/ FRA TANK. OGSAA VASK
SET PGM585_IND_T40  ; Z
LD TR0
AND PGM585_IND_T41_VALG  ; Z
ANDNOT C78_IND_VST80_K2  ; Z
ANDNOT T41_SPERR  ; SPERRER ALLE FUNKSJONER TIL/ FRA TANK. OGSAA VASK
SET PGM585_IND_T41  ; Z
; rung 14: INDIVID-RESET
LDNOT PGM585_START  ; Z
RSET PGM585_IND_T40  ; Z
RSET PGM585_IND_T41  ; Z
; rung 15: INDIVID-INNE INDIVID  ER VALGT
LDNOT PGM585_IND_T40  ; Z
ANDNOT PGM585_IND_T41  ; Z
OUTNOT PGM585_IND_INNE  ; Z
; rung 16: UTKOBLING-FORR UTKOBLING AV ALL SIKKERHET I PROGRAMMET MED UNTAK AV GJENSIDIGHETER I FORBINDELSE MED LØYPER
LD P_On
OUT TR0
AND=L(301) MANUELL_KOMMAND &1058508  ; KOMMANDOORD FOR IKKE LINJEKOMMANDOER
SET PGM585_TMU
LD TR0
AND PGM585_TMU
ANDNOT PGM585_START  ; Z
TIM 0785 #600  ; MAX-TID TMU OM IKKE LINJE LEGGES
LD TR0
LD=L(301) MANUELL_KOMMAND &2058508  ; KOMMANDOORD FOR IKKE LINJEKOMMANDOER
%OR PGM585_START  ; Z
OR PGM585_TMU_TID_S  ; MAX-TID TMU OM IKKE LINJE LEGGES
ANDLD
RSET PGM585_TMU

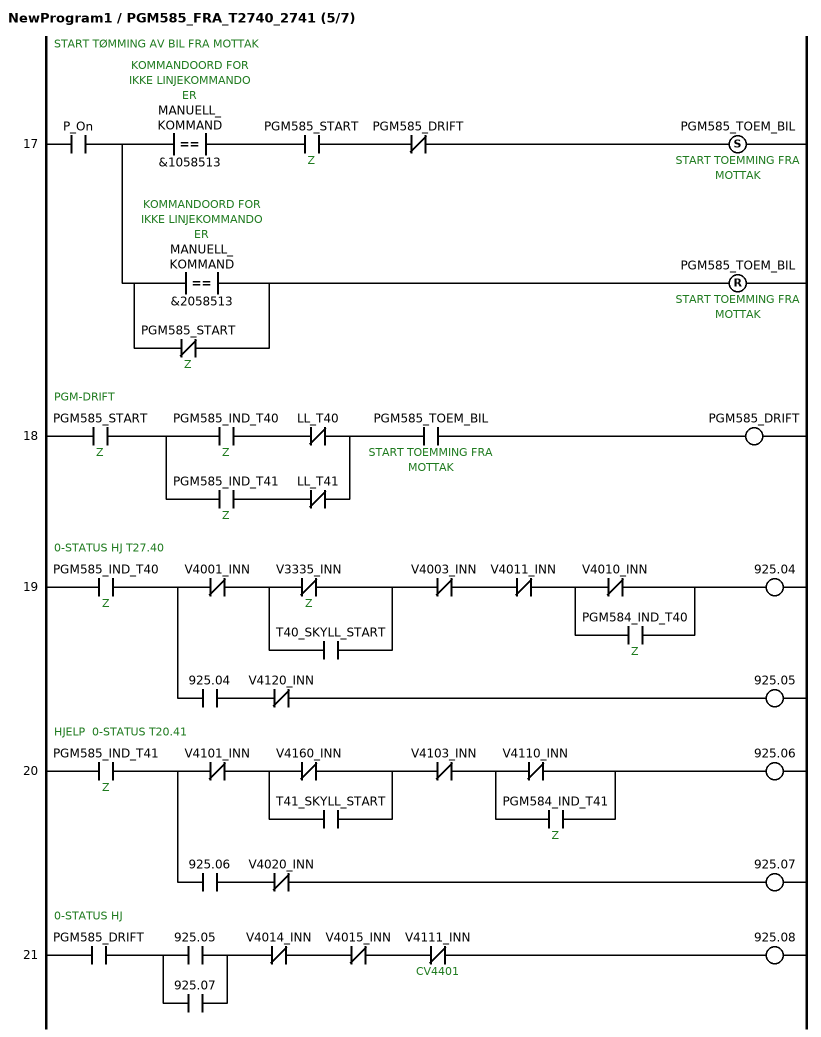
; rung 17: START TØMMING AV BIL FRA MOTTAK
LD P_On
OUT TR0
AND=L(301) MANUELL_KOMMAND &1058513  ; KOMMANDOORD FOR IKKE LINJEKOMMANDOER
AND PGM585_START  ; Z
ANDNOT PGM585_DRIFT
SET PGM585_TOEM_BIL  ; START TOEMMING FRA MOTTAK
LD TR0
LD=L(301) MANUELL_KOMMAND &2058513  ; KOMMANDOORD FOR IKKE LINJEKOMMANDOER
ORNOT PGM585_START  ; Z
ANDLD
RSET PGM585_TOEM_BIL  ; START TOEMMING FRA MOTTAK
; rung 18: PGM-DRIFT
LD PGM585_START  ; Z
LD PGM585_IND_T40  ; Z
ANDNOT LL_T40
LD PGM585_IND_T41  ; Z
ANDNOT LL_T41
ORLD
ANDLD
AND PGM585_TOEM_BIL  ; START TOEMMING FRA MOTTAK
OUT PGM585_DRIFT
; rung 19: 0-STATUS HJ T27.40
LD PGM585_IND_T40  ; Z
OUT TR0
ANDNOT V4001_INN
LDNOT V3335_INN  ; Z
OR T40_SKYLL_START
ANDLD
ANDNOT V4003_INN
ANDNOT V4011_INN
LDNOT V4010_INN
OR PGM584_IND_T40  ; Z
ANDLD
OUT 925.04
LD TR0
AND 925.04
ANDNOT V4120_INN
OUT 925.05
; rung 20: HJELP  0-STATUS T20.41
LD PGM585_IND_T41  ; Z
OUT TR0
ANDNOT V4101_INN
LDNOT V4160_INN
OR T41_SKYLL_START
ANDLD
ANDNOT V4103_INN
LDNOT V4110_INN
OR PGM584_IND_T41  ; Z
ANDLD
OUT 925.06
LD TR0
AND 925.06
ANDNOT V4020_INN
OUT 925.07
; rung 21: 0-STATUS HJ
LD PGM585_DRIFT
LD 925.05
OR 925.07
ANDLD
ANDNOT V4014_INN
ANDNOT V4015_INN
ANDNOT V4111_INN  ; CV4401
OUT 925.08

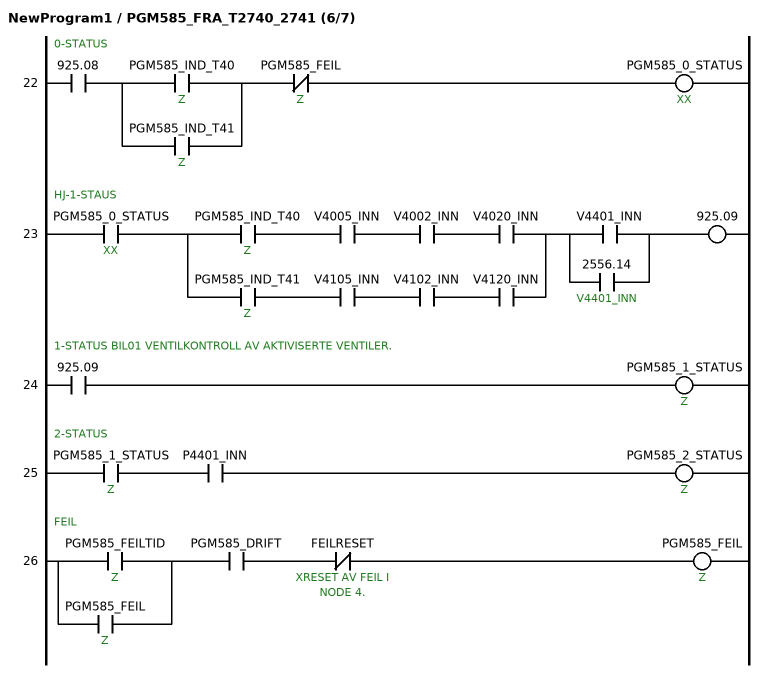
; rung 22: 0-STATUS
LD 925.08
LD PGM585_IND_T40  ; Z
OR PGM585_IND_T41  ; Z
ANDLD
ANDNOT PGM585_FEIL  ; Z
OUT PGM585_0_STATUS  ; XX
; rung 23: HJ-1-STAUS
LD PGM585_0_STATUS  ; XX
LD PGM585_IND_T40  ; Z
AND V4005_INN
AND V4002_INN
AND V4020_INN
LD PGM585_IND_T41  ; Z
AND V4105_INN
AND V4102_INN
AND V4120_INN
ORLD
ANDLD
LD V4401_INN
OR 2556.14  ; V4401_INN
ANDLD
OUT 925.09
; rung 24: 1-STATUS BIL01 VENTILKONTROLL AV AKTIVISERTE VENTILER.
LD 925.09
OUT PGM585_1_STATUS  ; Z
; rung 25: 2-STATUS
LD PGM585_1_STATUS  ; Z
AND P4401_INN
OUT PGM585_2_STATUS  ; Z
; rung 26: FEIL
LD PGM585_FEILTID  ; Z
OR PGM585_FEIL  ; Z
AND PGM585_DRIFT
ANDNOT FEILRESET  ; XRESET AV FEIL I NODE 4.
OUT PGM585_FEIL  ; Z

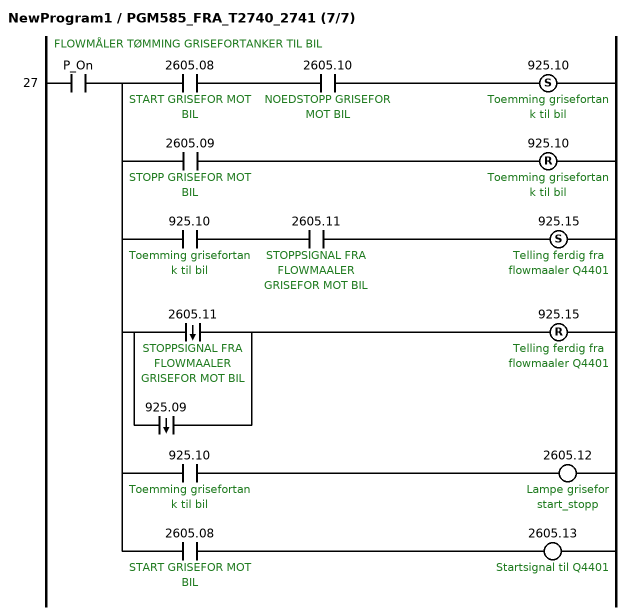
; rung 27: FLOWMÅLER TØMMING GRISEFORTANKER TIL BIL
LD P_On
OUT TR0
AND 2605.08  ; START GRISEFOR MOT BIL
AND 2605.10  ; NOEDSTOPP GRISEFOR MOT BIL
SET 925.10  ; Toemming grisefortank til bil
LD TR0
AND 2605.09  ; STOPP GRISEFOR MOT BIL
RSET 925.10  ; Toemming grisefortank til bil
LD TR0
AND 925.10  ; Toemming grisefortank til bil
AND 2605.11  ; STOPPSIGNAL FRA FLOWMAALER GRISEFOR MOT BIL
SET 925.15  ; Telling ferdig fra flowmaaler Q4401
LD TR0
%LD 2605.11  ; STOPPSIGNAL FRA FLOWMAALER GRISEFOR MOT BIL
%OR 925.09
ANDLD
RSET 925.15  ; Telling ferdig fra flowmaaler Q4401
LD TR0
AND 925.10  ; Toemming grisefortank til bil
OUT 2605.12  ; Lampe grisefor start_stopp
LD TR0
AND 2605.08  ; START GRISEFOR MOT BIL
OUT 2605.13  ; Startsignal til Q4401

### Section PGM586_ØKO_PASTEURER

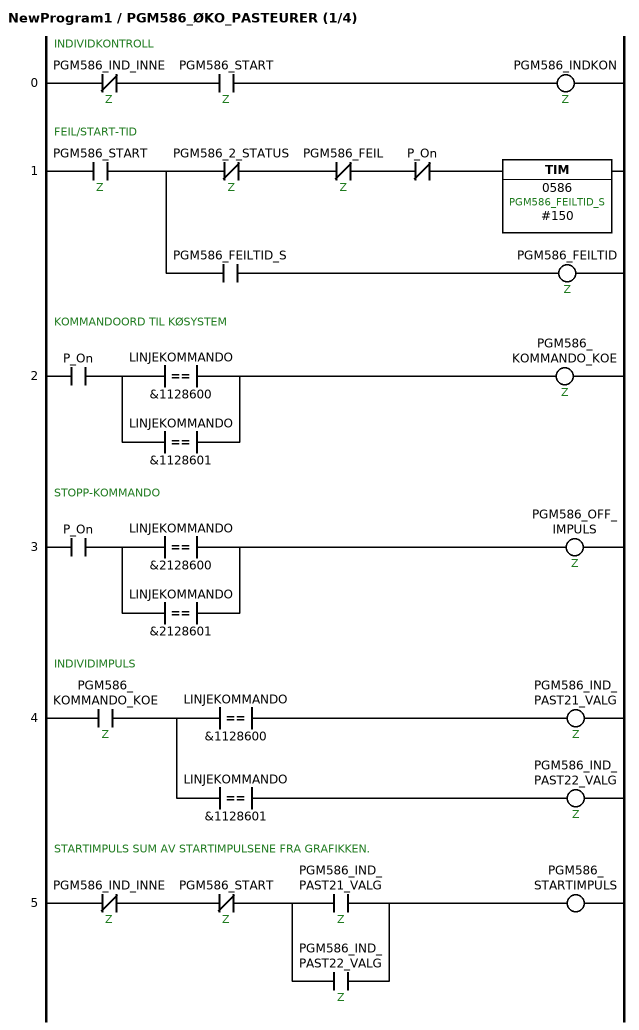
; rung 0: INDIVIDKONTROLL
LDNOT PGM586_IND_INNE  ; Z
AND PGM586_START  ; Z
OUT PGM586_INDKON  ; Z
; rung 1: FEIL/START-TID
LD PGM586_START  ; Z
OUT TR0
ANDNOT PGM586_2_STATUS  ; Z
ANDNOT PGM586_FEIL  ; Z
ANDNOT P_On
TIM 0586 #150  ; PGM586_FEILTID_S
LD TR0
AND PGM586_FEILTID_S
OUT PGM586_FEILTID  ; Z
; rung 2: KOMMANDOORD TIL KØSYSTEM
LD P_On
LD=L(301) LINJEKOMMANDO &1128600
OR=L(301) LINJEKOMMANDO &1128601
ANDLD
OUT PGM586_KOMMANDO_KOE  ; Z
; rung 3: STOPP-KOMMANDO
LD P_On
LD=L(301) LINJEKOMMANDO &2128600
OR=L(301) LINJEKOMMANDO &2128601
ANDLD
OUT PGM586_OFF_IMPULS  ; Z
; rung 4: INDIVIDIMPULS
LD PGM586_KOMMANDO_KOE  ; Z
OUT TR0
AND=L(301) LINJEKOMMANDO &1128600
OUT PGM586_IND_PAST21_VALG  ; Z
LD TR0
AND=L(301) LINJEKOMMANDO &1128601
OUT PGM586_IND_PAST22_VALG  ; Z
; rung 5: STARTIMPULS SUM AV STARTIMPULSENE FRA GRAFIKKEN.
LDNOT PGM586_IND_INNE  ; Z
ANDNOT PGM586_START  ; Z
LD PGM586_IND_PAST21_VALG  ; Z
OR PGM586_IND_PAST22_VALG  ; Z
ANDLD
OUT PGM586_STARTIMPULS

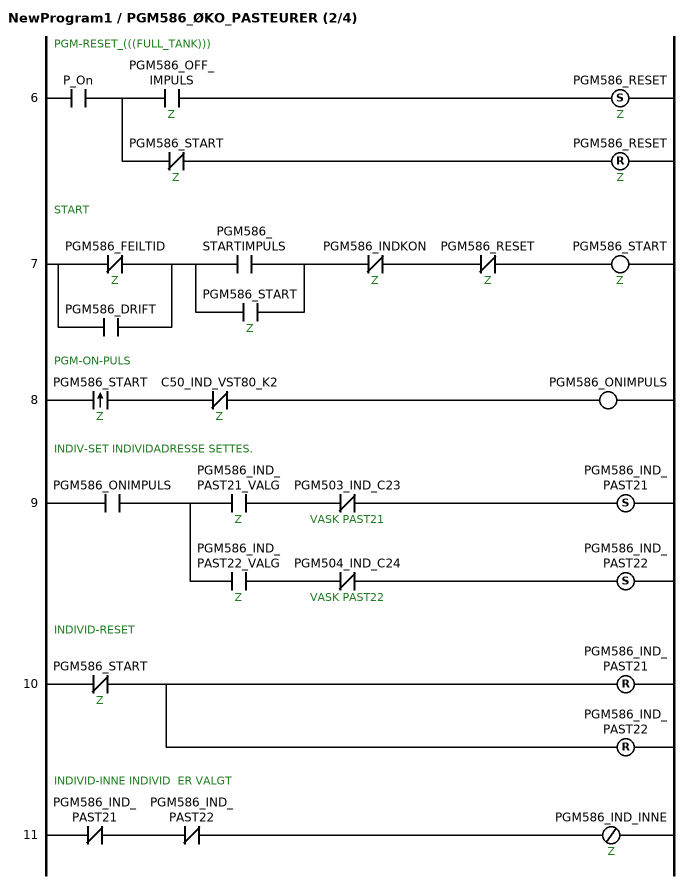
; rung 6: PGM-RESET_(((FULL_TANK)))
LD P_On
OUT TR0
AND PGM586_OFF_IMPULS  ; Z
SET PGM586_RESET  ; Z
LD TR0
ANDNOT PGM586_START  ; Z
RSET PGM586_RESET  ; Z
; rung 7: START
LDNOT PGM586_FEILTID  ; Z
OR PGM586_DRIFT
LD PGM586_STARTIMPULS
OR PGM586_START  ; Z
ANDLD
ANDNOT PGM586_INDKON  ; Z
ANDNOT PGM586_RESET  ; Z
OUT PGM586_START  ; Z
; rung 8: PGM-ON-PULS
@LD PGM586_START  ; Z
ANDNOT C50_IND_VST80_K2  ; Z
OUT PGM586_ONIMPULS
; rung 9: INDIV-SET INDIVIDADRESSE SETTES.
LD PGM586_ONIMPULS
OUT TR0
AND PGM586_IND_PAST21_VALG  ; Z
ANDNOT PGM503_IND_C23  ; VASK PAST21
SET PGM586_IND_PAST21
LD TR0
AND PGM586_IND_PAST22_VALG  ; Z
ANDNOT PGM504_IND_C24  ; VASK PAST22
SET PGM586_IND_PAST22
; rung 10: INDIVID-RESET
LDNOT PGM586_START  ; Z
RSET PGM586_IND_PAST21
RSET PGM586_IND_PAST22
; rung 11: INDIVID-INNE INDIVID  ER VALGT
LDNOT PGM586_IND_PAST21
ANDNOT PGM586_IND_PAST22
OUTNOT PGM586_IND_INNE  ; Z

